ABB RobotStudio station: multimove_python_20220504-124635.rsstn

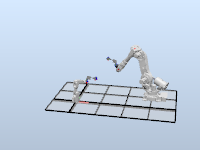
Station multimove_python (saved by RobotStudio 21.4.9700.0)
Controller MultiMove_python
  mechanical unit ROB_1: IRB1200_5_90_STD_03, 6 joints, base frame (0, 0, 0) mm
  mechanical unit ROB_2: IRB6640_180_255__04, 6 joints, base frame (3000, 1000, 0) mm, rotated rx 0 ry 0 rz 180 deg
Layout (positions relative to the parent item):
  - IRB1200_5_90_STD_03 [mechanism, from Robots\IRB1200_5_90_STD_03.rslib] at (0, 0, 0) mm; joint values [0.8857, -0.0016, 0.2585, 0.9299, -1.3596, -1.1212] (rad or m)
  - IRB6640_180_255__04 [mechanism, from Robots\IRB6640_180_255_G_04.rslib] at (3000, 1000, 0) mm, rotated rx 0 ry 0 rz 180 deg; joint values [-0.4372, 0.4636, 0.4396, -0.2373, -1.6421, 0.1232] (rad or m)
  - MyNewTool [mechanism, from models\Paintgun.rslib] at (350.28, 327.11, 815.16) mm, rotated rx 0.45 ry 59.18 rz -14.59 deg
  - MyNewTool_2 [mechanism, from models\Paintgun.rslib] at (1341.68, 1723.27, 1099.34) mm, rotated rx -4.66 ry 48.83 rz 166.88 deg
Attachment: MyNewTool is attached to IRB1200_5_90_STD_03 / Link6
Attachment: MyNewTool_2 is attached to IRB6640_180_255__04 / Link6
Targets, tools, work objects and paths stored in the station, written as RAPID:
! task T_ROB1
MODULE CalibData
  PERS tooldata MyNewTool:=[TRUE,[[50,0,450],[1,0,0,0]],[1,[0,0,1],[1,0,0,0],0,0,0]];
ENDMODULE

! task T_ROB2
MODULE CalibData
  PERS tooldata MyNewTool:=[TRUE,[[50,0,450],[1,0,0,0]],[1,[0,0,1],[1,0,0,0],0,0,0]];
ENDMODULE

